// TIA Portal V19 export
VAR_GLOBAL   // PLC tag table "Default tag table_1"
   Tag_3 AT %M0.1 : Bool;
END_VAR
